PROGRAM MAIN
VAR
END_VAR

END_PROGRAM

(* stored: Version 1.1.0.1
   POU MAIN: Id {a67776c6-7921-42f7-b7a7-80948cc46fac} *)
